Fanuc KAREL source: kb00001.KL

-- PROVISIONAL review KL for V940-1; original PC SHA256 2579f349a6665a2069981512503bade0f0dc6378985d1628b66a0a64bd5cd2a0
-- Incomplete behavior may be omitted. Consult companion uncertainty JSON. Do not deploy.
PROGRAM KB00001
%NOLOCKGROUP
BEGIN
  -- V9_ZERO_TABLE_METADATA_HINT layout=0002_ascii; no indexed target words; source/name/runtime held
  -- UNRESOLVED_PC offsets 5-14; opcodes 3F,75
  -- UNRESOLVED_PC offsets 19-26; opcodes 9D,23
  -- UNRESOLVED_PC offsets 31-38; opcodes 9D,23
  -- UNRESOLVED_PC offsets 43-50; opcodes 9D,23
  -- UNRESOLVED_PC offsets 55-85; opcodes 27,22,2A,22,22,22,31
  -- UNRESOLVED_PC offsets 90-94; opcodes 7F
END KB00001
